FUNCTION_BLOCK Test_ReadBySymbolName EXTENDS T_UnitTestBase
VAR
    AdsReadBySymbolName : T_AdsReadBySymbolName;
    ValueToRead : INT;
    ReadResult  : INT;
    ScanCount : DINT;
    State: INT;
END_VAR

CASE State OF
    0:
        ValueToRead := 1234;
        ReadResult := 0;
        ScanCount := 0;
    
        AdsReadBySymbolName.Execute(
            AmsNetId:= '', 
            Port:= Constants.PortNo, 
            SymbolName:= 'PB_TestRunner.Test_ReadBySymbolName.ValueToRead', 
            ReadDataAddress:= ADR(ReadResult), 
            ReadDataLength:= SIZEOF(ReadResult), 
            KeepSymbolHandle:= FALSE);

        State := 10;
        
    10:
        ScanCount := ScanCount + 1;
        IF NOT AdsReadBySymbolName.Execution.Busy THEN
            State := 20;    
		END_IF
        
    20:
        Assertion.AssertEquals_INT(
            Expected     := 1234,
            Actual       := ReadResult,
            Variablename := 'ReadResult'); 
 
        TestFinished();
        State := 0;
END_CASE

AdsReadBySymbolName();

END_FUNCTION_BLOCK

(* stored: Version 1.1.0.1, ProductVersion 3.1.4024.4
   POU Test_ReadBySymbolName: Id {30924da5-0ef2-00c1-3fa5-f920c6036a59}, SpecialFunc None *)
